FUNCTION_BLOCK FB_LogLevel		// Helper for setting and getting ENUM as string
VAR
	level:	E_LOG_LEVEL;
END_VAR

METHOD PUBLIC asString : T_DEFAULT_STR
CASE level OF
	E_LOG_LEVEL.TRACE:
		asString := '[TRACE]';
	
	E_LOG_LEVEL.DEBUG:
		asString := '[DEBUG]';
	
	E_LOG_LEVEL.INFO:
		asString := '[INFO]';
	
	E_LOG_LEVEL.WARN:
		asString := '[WARN]';
	
	E_LOG_LEVEL.ERROR:
		asString := '[ERROR]';

	E_LOG_LEVEL.OFF:
		asString := 'do not use this log level';

ELSE
	asString := 'todo';
END_CASE
END_METHOD

METHOD public set : BOOL
VAR_INPUT
	iLevel:	E_LOG_LEVEL;
END_VAR
level := iLevel;
END_METHOD

END_FUNCTION_BLOCK

(* stored: Version 1.1.0.1, ProductVersion 3.1.4026.18
   POU FB_LogLevel: Id {ba3a63a2-bb7c-46bd-8653-829240b48843}, SpecialFunc None
   Method asString: Id {24937936-5e39-47f2-8f82-6be5d6045ac9}
   Method set: Id {c6324bcb-4808-4dd3-b9f2-5fc557d9b851} *)
